INTERFACE I_Station

METHOD Clear : BOOL
VAR_INPUT
END_VAR
END_METHOD

METHOD Enable : BOOL
VAR_INPUT
END_VAR
END_METHOD

PROPERTY InPosition : BOOL
GET
END_GET
END_PROPERTY

METHOD JobDone : BOOL
VAR_INPUT
END_VAR
END_METHOD

METHOD SetPosAttractStep : BOOL
VAR_INPUT
	step : INT;
END_VAR
END_METHOD

METHOD SetPosMoverStep : BOOL
VAR_INPUT
	posIndex	: INT;
	step		: INT;
END_VAR
END_METHOD

END_INTERFACE

(* stored: Version 1.1.0.1
   Itf I_Station: Id {3b7371aa-5b61-48d8-b861-536b44e57f57}
   Method Clear: Id {593d480f-37ab-4907-8156-54c4317194a7}
   Method Enable: Id {cd149905-4a43-4593-a4f6-19abdb693ea9}
   Property InPosition: Id {f2d4b04b-b370-4fe7-b85d-25115261eea8}
   Get Get: Id {ebf3a048-7cf1-4b73-8cd4-b432d8bca665}
   Method JobDone: Id {6c7e61b6-6f99-4381-8683-bb2460e8382d}
   Method SetPosAttractStep: Id {0ca5243e-e31c-498d-a259-e2d991574f21}
   Method SetPosMoverStep: Id {8c27bf90-a502-47af-a4e1-258c5da5ca9e} *)
